{attribute 'qualified_only'}
VAR_GLOBAL
END_VAR

(* stored: Version 1.1.0.1, ProductVersion 3.1.4024.12
   GVL G_Parameters: Id {ce2e188f-b995-4eeb-a43c-5106c94f1d2b} *)
